FUNCTION_BLOCK S7_READ_CONTINUOUS_SOLDERING
  {SET_ATTRIBUTE(OpcUa, DEVICE.SENSOR)}
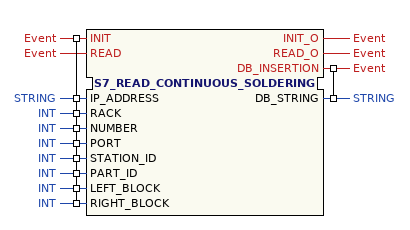
  EVENT_INPUT
    INIT WITH IP_ADDRESS, RACK, NUMBER, PORT, STATION_ID, PART_ID, LEFT_BLOCK, RIGHT_BLOCK;
    READ;
  END_EVENT
  EVENT_OUTPUT
    INIT_O;
    READ_O;
    DB_INSERTION WITH DB_STRING;
  END_EVENT
  VAR_INPUT
    IP_ADDRESS : STRING; {SET_ATTRIBUTE(OpcUa, Constant.RUN)}
    RACK : INT; {SET_ATTRIBUTE(OpcUa, Constant.RUN)}
    NUMBER : INT; {SET_ATTRIBUTE(OpcUa, Constant.RUN)}
    PORT : INT; {SET_ATTRIBUTE(OpcUa, Constant.RUN)}
    STATION_ID : INT; {SET_ATTRIBUTE(OpcUa, Constant.RUN)}
    PART_ID : INT; {SET_ATTRIBUTE(OpcUa, Constant.RUN)}
    LEFT_BLOCK : INT; {SET_ATTRIBUTE(OpcUa, Constant.RUN)}
    RIGHT_BLOCK : INT; {SET_ATTRIBUTE(OpcUa, Constant.RUN)}
  END_VAR
  VAR_OUTPUT
    DB_STRING : STRING; {SET_ATTRIBUTE(OpcUa, Variable.RUN)}
  END_VAR
END_FUNCTION_BLOCK
